PROGRAM MAIN
VAR
END_VAR

END_PROGRAM

(* stored: Version 1.1.0.1, ProductVersion 3.1.4024.10
   POU MAIN: Id {aefaa972-af2a-4a47-917d-7a351e8d118b}, SpecialFunc None *)
